% RSLogix 500 project Inventory Management.RSS, saved by version 8.30.00.16 %
PROJECT "UNTITLED"    % processor: Bul.1763 MicroLogix 1100 Series B %

PROGRAM FILES
  LAD 2   16 rungs

DATA FILES
  O0 OUTPUT  4 elements
  I1 INPUT  6 elements
  S2 STATUS  66 elements
  B3 BINARY  2 elements
  T4 TIMER  1 elements
  C5 COUNTER  1 elements
  R6 CONTROL  1 elements
  N7 INTEGER  9 elements
  F8 FLOAT  1 elements
  ST9 STRING  6 elements

LADDER 2
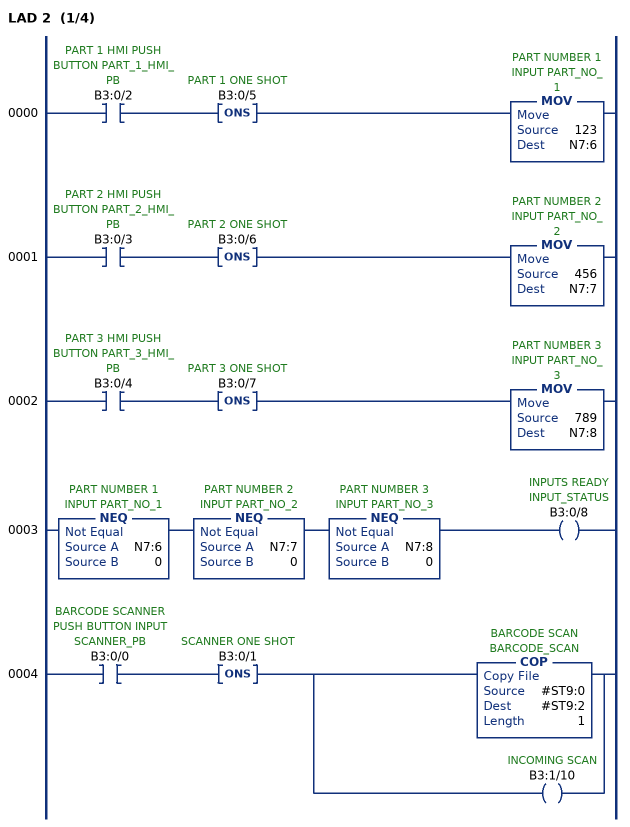
% Rung: 0 %
SOR XIC B3:0/2 ONS B3:0/5 MOV 123 N7:6 EOR
%   B3:0/2  PART_1_HMI_PB  "PART 1 HMI PUSH BUTTON" %
%   B3:0/5  "PART 1 ONE SHOT" %
%   N7:6  PART_NO_1  "PART NUMBER 1 INPUT" %
% Rung: 1 %
SOR XIC B3:0/3 ONS B3:0/6 MOV 456 N7:7 EOR
%   B3:0/3  PART_2_HMI_PB  "PART 2 HMI PUSH BUTTON" %
%   B3:0/6  "PART 2 ONE SHOT" %
%   N7:7  PART_NO_2  "PART NUMBER 2 INPUT" %
% Rung: 2 %
SOR XIC B3:0/4 ONS B3:0/7 MOV 789 N7:8 EOR
%   B3:0/4  PART_3_HMI_PB  "PART 3 HMI PUSH BUTTON" %
%   B3:0/7  "PART 3 ONE SHOT" %
%   N7:8  PART_NO_3  "PART NUMBER 3 INPUT" %
% Rung: 3 %
SOR NEQ N7:6 0 NEQ N7:7 0 NEQ N7:8 0 OTE B3:0/8 EOR
%   N7:6  PART_NO_1  "PART NUMBER 1 INPUT" %
%   N7:7  PART_NO_2  "PART NUMBER 2 INPUT" %
%   N7:8  PART_NO_3  "PART NUMBER 3 INPUT" %
%   B3:0/8  INPUT_STATUS  "INPUTS READY" %
% Rung: 4 %
SOR XIC B3:0/0 ONS B3:0/1 BST COP #ST9:0 #ST9:2 1 NXB OTE B3:1/10 BND EOR
%   B3:0/0  SCANNER_PB  "BARCODE SCANNER PUSH BUTTON INPUT" %
%   B3:0/1  "SCANNER ONE SHOT" %
%   ST9:2  BARCODE_SCAN  "BARCODE SCAN" %
%   B3:1/10  "INCOMING SCAN" %

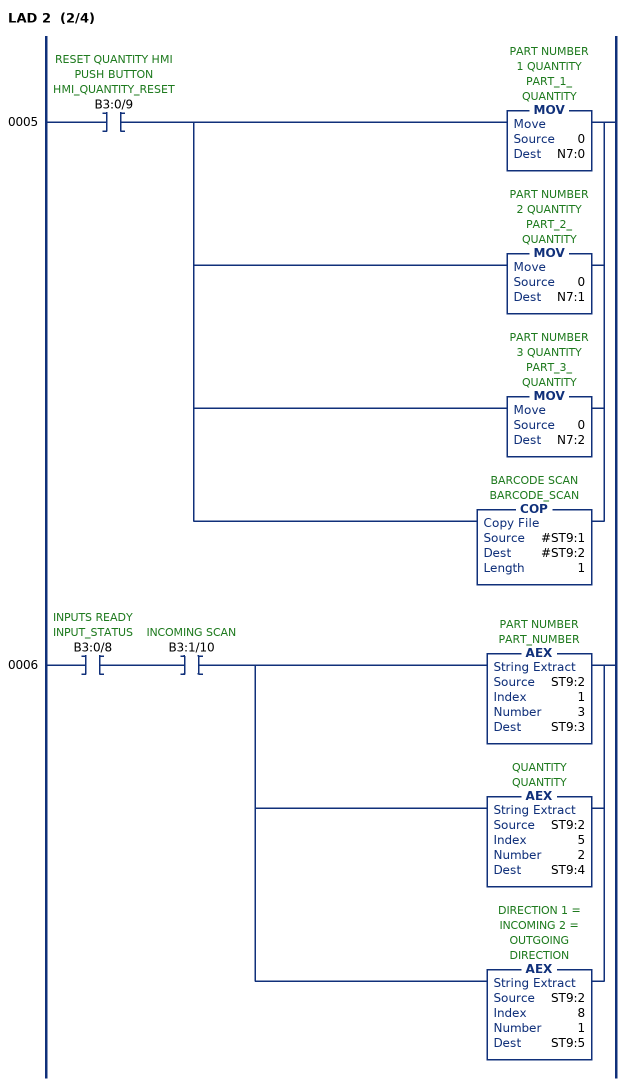
% Rung: 5 %
SOR XIC B3:0/9 BST MOV 0 N7:0 NXB MOV 0 N7:1 NXB MOV 0 N7:2 NXB COP #ST9:1 #ST9:2 1 BND EOR
%   B3:0/9  HMI_QUANTITY_RESET  "RESET QUANTITY HMI PUSH BUTTON" %
%   N7:0  PART_1_QUANTITY  "PART NUMBER 1 QUANTITY" %
%   N7:1  PART_2_QUANTITY  "PART NUMBER 2 QUANTITY" %
%   N7:2  PART_3_QUANTITY  "PART NUMBER 3 QUANTITY" %
%   ST9:1  "RESET STRING" %
%   ST9:2  BARCODE_SCAN  "BARCODE SCAN" %
% Rung: 6 %
SOR XIC B3:0/8 XIC B3:1/10 BST AEX ST9:2 1 3 ST9:3 NXB AEX ST9:2 5 2 ST9:4 NXB AEX ST9:2 8 1 ST9:5 BND EOR
%   B3:0/8  INPUT_STATUS  "INPUTS READY" %
%   B3:1/10  "INCOMING SCAN" %
%   ST9:2  BARCODE_SCAN  "BARCODE SCAN" %
%   ST9:3  PART_NUMBER  "PART NUMBER" %
%   ST9:4  QUANTITY  "QUANTITY" %
%   ST9:5  DIRECTION  "DIRECTION 1 = INCOMING 2 = OUTGOING" %

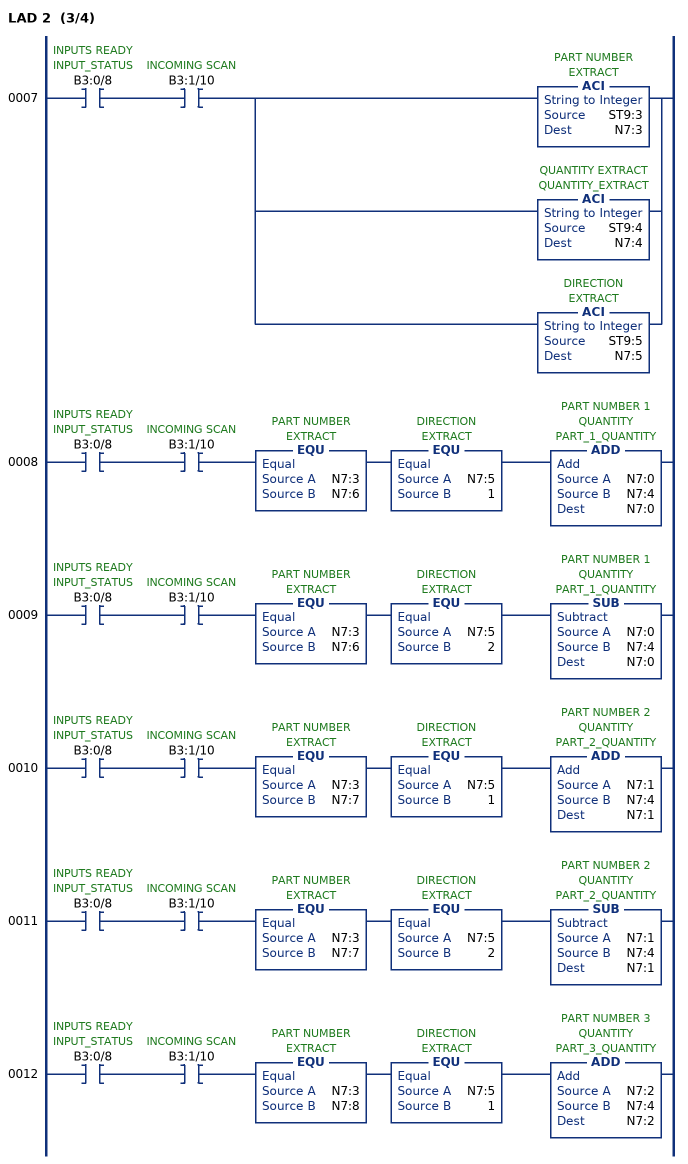
% Rung: 7 %
SOR XIC B3:0/8 XIC B3:1/10 BST ACI ST9:3 N7:3 NXB ACI ST9:4 N7:4 NXB ACI ST9:5 N7:5 BND EOR
%   B3:0/8  INPUT_STATUS  "INPUTS READY" %
%   B3:1/10  "INCOMING SCAN" %
%   ST9:3  PART_NUMBER  "PART NUMBER" %
%   N7:3  "PART NUMBER EXTRACT" %
%   ST9:4  QUANTITY  "QUANTITY" %
%   N7:4  QUANTITY_EXTRACT  "QUANTITY EXTRACT" %
%   ST9:5  DIRECTION  "DIRECTION 1 = INCOMING 2 = OUTGOING" %
%   N7:5  "DIRECTION EXTRACT" %
% Rung: 8 %
SOR XIC B3:0/8 XIC B3:1/10 EQU N7:3 N7:6 EQU N7:5 1 ADD N7:0 N7:4 N7:0 EOR
%   B3:0/8  INPUT_STATUS  "INPUTS READY" %
%   B3:1/10  "INCOMING SCAN" %
%   N7:3  "PART NUMBER EXTRACT" %
%   N7:6  PART_NO_1  "PART NUMBER 1 INPUT" %
%   N7:5  "DIRECTION EXTRACT" %
%   N7:0  PART_1_QUANTITY  "PART NUMBER 1 QUANTITY" %
%   N7:4  QUANTITY_EXTRACT  "QUANTITY EXTRACT" %
% Rung: 9 %
SOR XIC B3:0/8 XIC B3:1/10 EQU N7:3 N7:6 EQU N7:5 2 SUB N7:0 N7:4 N7:0 EOR
%   B3:0/8  INPUT_STATUS  "INPUTS READY" %
%   B3:1/10  "INCOMING SCAN" %
%   N7:3  "PART NUMBER EXTRACT" %
%   N7:6  PART_NO_1  "PART NUMBER 1 INPUT" %
%   N7:5  "DIRECTION EXTRACT" %
%   N7:0  PART_1_QUANTITY  "PART NUMBER 1 QUANTITY" %
%   N7:4  QUANTITY_EXTRACT  "QUANTITY EXTRACT" %
% Rung: 10 %
SOR XIC B3:0/8 XIC B3:1/10 EQU N7:3 N7:7 EQU N7:5 1 ADD N7:1 N7:4 N7:1 EOR
%   B3:0/8  INPUT_STATUS  "INPUTS READY" %
%   B3:1/10  "INCOMING SCAN" %
%   N7:3  "PART NUMBER EXTRACT" %
%   N7:7  PART_NO_2  "PART NUMBER 2 INPUT" %
%   N7:5  "DIRECTION EXTRACT" %
%   N7:1  PART_2_QUANTITY  "PART NUMBER 2 QUANTITY" %
%   N7:4  QUANTITY_EXTRACT  "QUANTITY EXTRACT" %
% Rung: 11 %
SOR XIC B3:0/8 XIC B3:1/10 EQU N7:3 N7:7 EQU N7:5 2 SUB N7:1 N7:4 N7:1 EOR
%   B3:0/8  INPUT_STATUS  "INPUTS READY" %
%   B3:1/10  "INCOMING SCAN" %
%   N7:3  "PART NUMBER EXTRACT" %
%   N7:7  PART_NO_2  "PART NUMBER 2 INPUT" %
%   N7:5  "DIRECTION EXTRACT" %
%   N7:1  PART_2_QUANTITY  "PART NUMBER 2 QUANTITY" %
%   N7:4  QUANTITY_EXTRACT  "QUANTITY EXTRACT" %
% Rung: 12 %
SOR XIC B3:0/8 XIC B3:1/10 EQU N7:3 N7:8 EQU N7:5 1 ADD N7:2 N7:4 N7:2 EOR
%   B3:0/8  INPUT_STATUS  "INPUTS READY" %
%   B3:1/10  "INCOMING SCAN" %
%   N7:3  "PART NUMBER EXTRACT" %
%   N7:8  PART_NO_3  "PART NUMBER 3 INPUT" %
%   N7:5  "DIRECTION EXTRACT" %
%   N7:2  PART_3_QUANTITY  "PART NUMBER 3 QUANTITY" %
%   N7:4  QUANTITY_EXTRACT  "QUANTITY EXTRACT" %

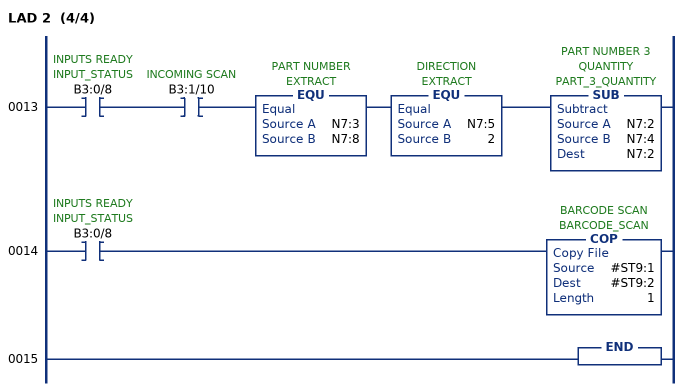
% Rung: 13 %
SOR XIC B3:0/8 XIC B3:1/10 EQU N7:3 N7:8 EQU N7:5 2 SUB N7:2 N7:4 N7:2 EOR
%   B3:0/8  INPUT_STATUS  "INPUTS READY" %
%   B3:1/10  "INCOMING SCAN" %
%   N7:3  "PART NUMBER EXTRACT" %
%   N7:8  PART_NO_3  "PART NUMBER 3 INPUT" %
%   N7:5  "DIRECTION EXTRACT" %
%   N7:2  PART_3_QUANTITY  "PART NUMBER 3 QUANTITY" %
%   N7:4  QUANTITY_EXTRACT  "QUANTITY EXTRACT" %
% Rung: 14 %
SOR XIC B3:0/8 COP #ST9:1 #ST9:2 1 EOR
%   B3:0/8  INPUT_STATUS  "INPUTS READY" %
%   ST9:1  "RESET STRING" %
%   ST9:2  BARCODE_SCAN  "BARCODE SCAN" %
% Rung: 15 %
SOR END EOR
